// Mitsubishi GX Works2 project: group24_exe2   PLC: FX3G

// global labels: Global1
VAR_GLOBAL
  all_check AT M1 : BOOL;
  switch_check_start AT X007 : BOOL;
  start_day_lamp AT Y007 : BOOL;
  CREAM_CONTAINER AT D2006 : REAL;
  Cream_Transfer_Start AT X011 : BOOL;
  splash_bag AT D2010 : REAL;
  BISCUITS_CONTAINER AT D2012 : REAL;
  Tray AT D2014 : REAL;
  Start_Machine_A AT X010 : BOOL;
  System_On AT M0 : BOOL;
  Close_System AT X005 : BOOL;
  Splashing_System AT Y004 : BOOL;
  Sen1 AT X001 : BOOL;
  Sen4 AT X002 : BOOL;
  Sen30 AT X004 : BOOL;
  Sen15 AT X003 : BOOL;
  Timer_Out_1 AT TS1 : BOOL;
  Sirogin0 AT Y000 : BOOL;
  Sirogin1 AT Y001 : BOOL;
  First_T AT TC1 : BOOL;
  Second_T AT TC2 : BOOL;
  Timer_Out_2 AT TS2 : BOOL;
  Help_Start_1 AT M10 : BOOL;
  Help_Start_2 AT M11 : BOOL;
  Help_Start_3 AT M12 : BOOL;
  Evhov AT M40 : BOOL;
END_VAR
VAR_GLOBAL CONSTANT
  Time_For_Evhov : INT := 40;
END_VAR
VAR_GLOBAL
  start_chocolate AT X006 : BOOL;
END_VAR
VAR_GLOBAL CONSTANT
  input_1 : INT;
  input_5 : INT := 1995;
END_VAR
VAR_GLOBAL
  TC_4 AT TC4 : BOOL;
  Chocolate_Dip_Lamp AT Y003 : BOOL;
  TS_4 AT TS4 : BOOL;
  CRAMBO_PACKAGE_LIGHT AT Y002 : BOOL;
  CC_5 AT CC5 : BOOL;
END_VAR
VAR_GLOBAL CONSTANT
  Count_5 : INT := 5;
END_VAR
VAR_GLOBAL
  CS_5 AT CS5 : BOOL;
  START_PACKAGING AT X000 : BOOL;
  M14_STOP_LAMP AT M14 : BOOL;
END_VAR
VAR_GLOBAL CONSTANT
  Count_6 : INT := 6;
END_VAR
VAR_GLOBAL
  M16_lamp AT M16 : BOOL;
  CS_6 AT CS6 : BOOL;
  CC_6 AT CC6 : BOOL;
END_VAR
VAR_GLOBAL CONSTANT
  input_10 : INT := 4000;
END_VAR
VAR_GLOBAL
  analog_input_10 AT M20 : BOOL;
  analog_input_5 AT M18 : BOOL;
  Check_New_Iteration_Cream AT M24 : BOOL;
  Check_New_Iteration_chocolate AT M26 : BOOL;
  Check_New_Iteration_Biscuits AT M28 : BOOL;
  CHOCOLATE_CONTAINER AT D2022 : REAL;
  CHOCOLATE_DIPPING AT D2020 : REAL;
  TS_30 AT TS30 : BOOL;
  TC_30 AT TC30 : BOOL;
END_VAR
VAR_GLOBAL CONSTANT
  Three_sec : INT := 30;
END_VAR
VAR_GLOBAL
  helperhivhuv AT M9 : BOOL;
  Help_Lamp AT M2 : BOOL;
  analog_input_cream AT D2026 : REAL;
  analog_input_chocolat AT D2028 : REAL;
  analog_input_biscuit AT D2030 : REAL;
  Help_Lamp_On_1 AT M31 : BOOL;
  Help_Lamp_On_2 AT M32 : BOOL;
  Hivhiv_transport AT TC40 : BOOL;
  TS_40 AT TS40 : BOOL;
END_VAR
VAR_GLOBAL CONSTANT
  crembo_mul : REAL := 40;
  const_120 : REAL := 120;
  const_240 : REAL := 240;
  const_300 : REAL := 300;
  const_6 : REAL := 6;
END_VAR
VAR_GLOBAL
  finished_crembos AT D2018 : REAL;
  analogiNPUT AT D8280 : INT;
  save_analogiNPUT AT D2000 : INT;
END_VAR
VAR_GLOBAL CONSTANT
  hivhuv_Seconds : INT := 3;
END_VAR
VAR_GLOBAL
  finished_dipping AT M70 : BOOL;
END_VAR
VAR_GLOBAL CONSTANT
  Timer_For_Chocolate_Dipping : INT := 50;
END_VAR
VAR_GLOBAL
  analog_output AT D8282 : INT;
END_VAR

// task Task_01 (event TRUE, interval 0, priority 31): POU_01

PROGRAM POU_01
(* structured ladder/FBD written out as ST: instructions are called as NAME(EN, inputs, outputs); _pN, _eN, _tN stand for wires *)
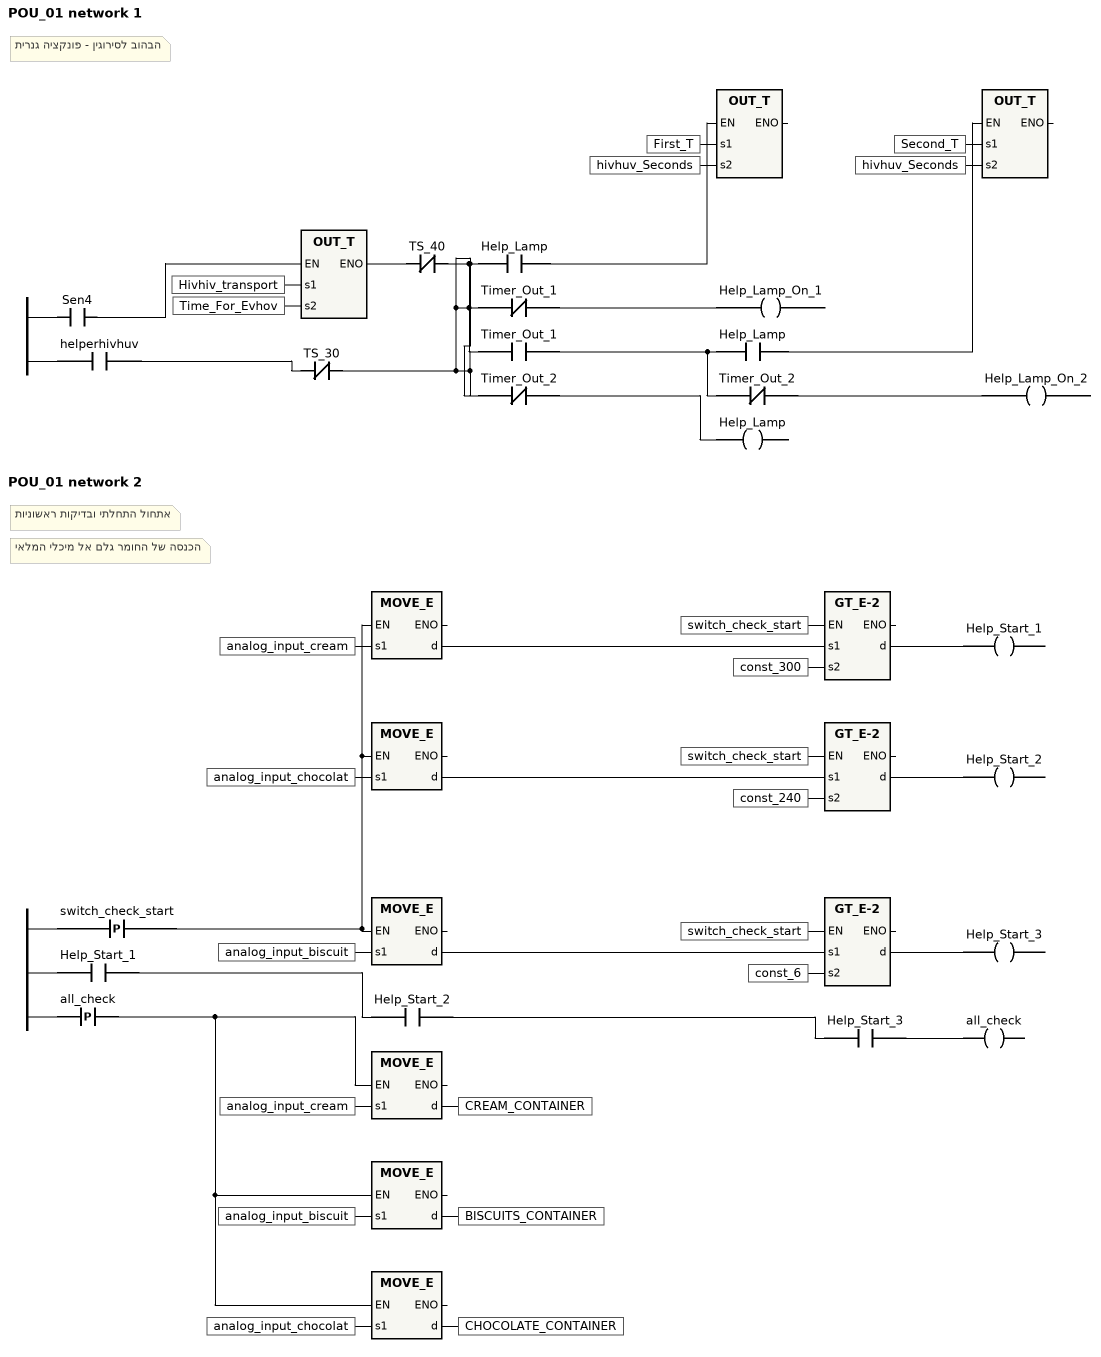
(* network 1 *)
(* הבהוב לסירוגין - פונקציה גנרית *)
_e1 := OUT_T(Sen4, Hivhiv_transport, Time_For_Evhov);
_p2 := (_e1 AND NOT TS_40) OR (helperhivhuv AND NOT TS_30);
OUT_T(_p2 AND Help_Lamp, First_T, hivhuv_Seconds);
Help_Lamp_On_1 := _p2 AND NOT Timer_Out_1;
_p3 := _p2 AND Timer_Out_1;
OUT_T(_p3 AND Help_Lamp, Second_T, hivhuv_Seconds);
Help_Lamp_On_2 := _p3 AND NOT Timer_Out_2;
Help_Lamp := _p2 AND NOT Timer_Out_2;
(* network 2 *)
(* אתחול התחלתי ובדיקות ראשוניות *)
(* הכנסה של החומר גלם אל מיכלי המלאי *)
_p1 := LDP(TRUE, switch_check_start);
MOVE_E(_p1, analog_input_cream, _t2);
GT_E(switch_check_start, _t2, const_300, _t3);
Help_Start_1 := _t3;
MOVE_E(_p1, analog_input_chocolat, _t4);
GT_E(switch_check_start, _t4, const_240, _t5);
Help_Start_2 := _t5;
MOVE_E(_p1, analog_input_biscuit, _t6);
GT_E(switch_check_start, _t6, const_6, _t7);
Help_Start_3 := _t7;
all_check := Help_Start_1 AND Help_Start_2 AND Help_Start_3;
_p8 := LDP(TRUE, all_check);
MOVE_E(_p8, analog_input_cream, CREAM_CONTAINER);
MOVE_E(_p8, analog_input_biscuit, BISCUITS_CONTAINER);
MOVE_E(_p8, analog_input_chocolat, CHOCOLATE_CONTAINER);
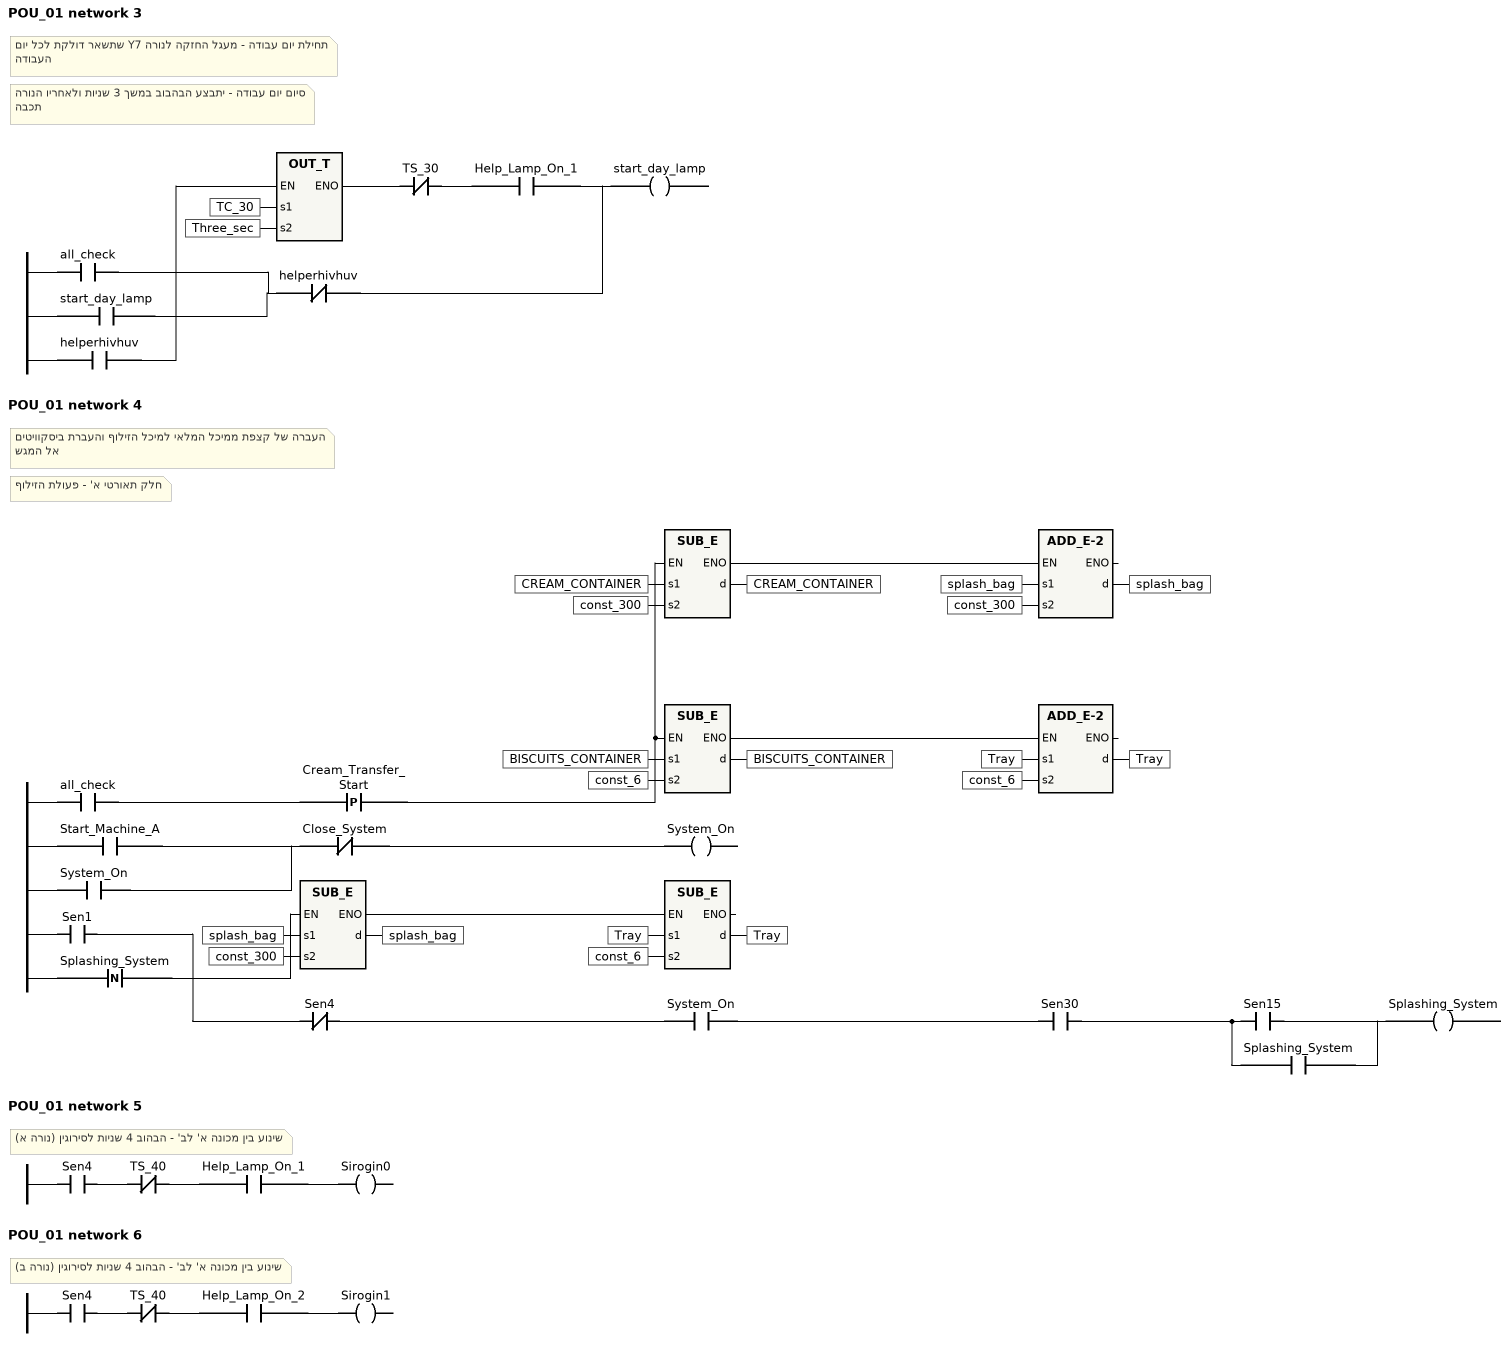
(* network 3 *)
(* תחילת יום עבודה - מעגל החזקה לנורה Y7 שתשאר דולקת לכל יום העבודה *)
(* סיום יום עבודה - יתבצע הבהבוב במשך 3 שניות ולאחריו הנורה תכבה *)
_e1 := OUT_T(helperhivhuv, TC_30, Three_sec);
start_day_lamp := ((all_check OR start_day_lamp) AND NOT helperhivhuv) OR (_e1 AND NOT TS_30 AND Help_Lamp_On_1);
(* network 4 *)
(* העברה של קצפת ממיכל המלאי למיכל הזילוף והעברת ביסקוויטים אל המגש *)
(* חלק תאורטי א' - פעולת הזילוף *)
_p1 := all_check AND LDP(TRUE, Cream_Transfer_Start);
_e2 := SUB_E(_p1, CREAM_CONTAINER, const_300, CREAM_CONTAINER);
ADD_E(_e2, splash_bag, const_300, splash_bag);
_e3 := SUB_E(_p1, BISCUITS_CONTAINER, const_6, BISCUITS_CONTAINER);
ADD_E(_e3, Tray, const_6, Tray);
System_On := (Start_Machine_A OR System_On) AND NOT Close_System;
_p4 := Sen1 AND NOT Sen4 AND System_On AND Sen30;
Splashing_System := (_p4 AND Sen15) OR (_p4 AND Splashing_System);
_e5 := SUB_E(LDF(TRUE, Splashing_System), splash_bag, const_300, splash_bag);
SUB_E(_e5, Tray, const_6, Tray);
(* network 5 *)
(* שינוע בין מכונה א' לב' - הבהוב 4 שניות לסירוגין (נורה א) *)
Sirogin0 := Sen4 AND NOT TS_40 AND Help_Lamp_On_1;
(* network 6 *)
(* שינוע בין מכונה א' לב' - הבהוב 4 שניות לסירוגין (נורה ב) *)
Sirogin1 := Sen4 AND NOT TS_40 AND Help_Lamp_On_2;
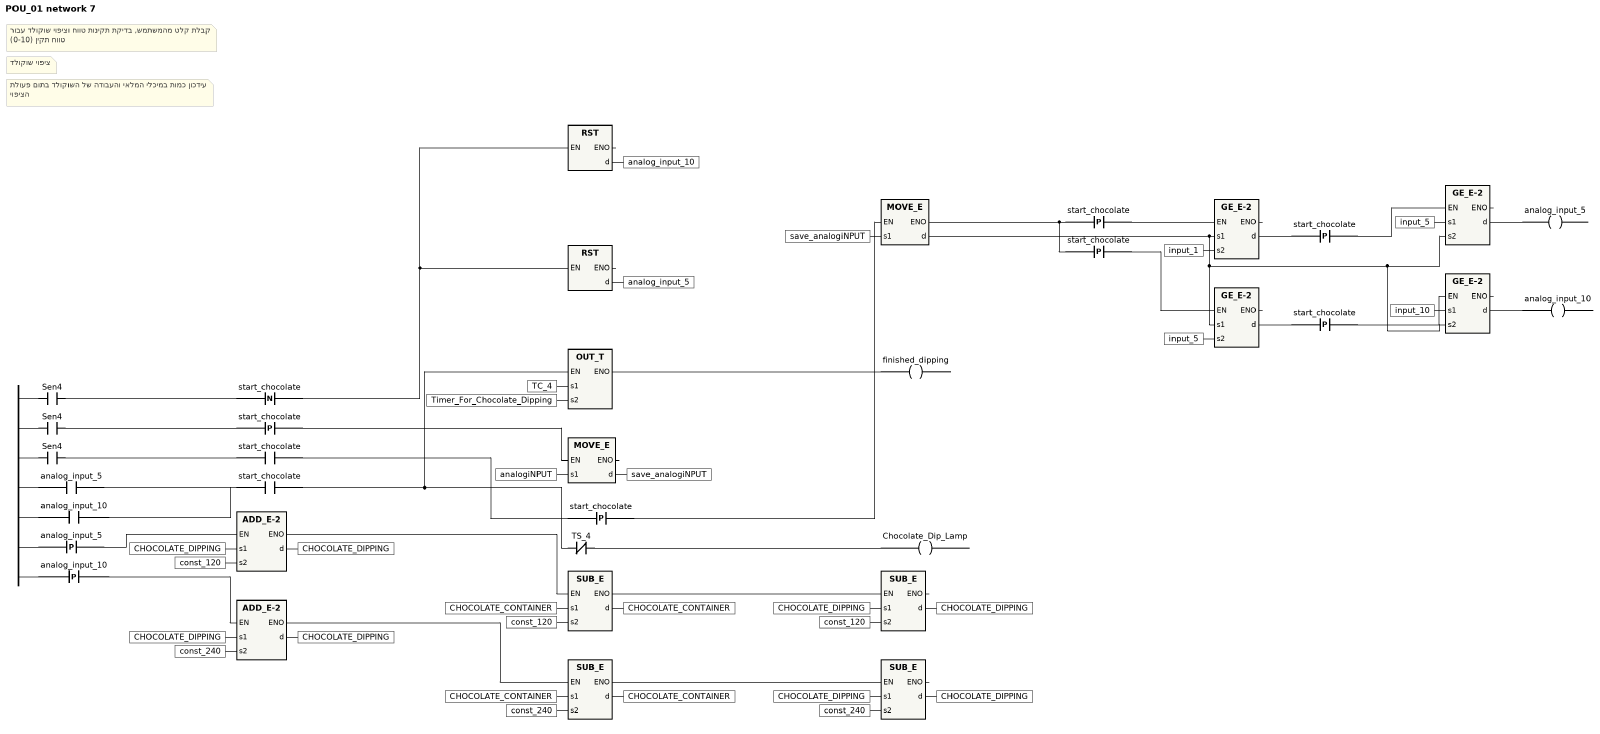
(* network 7 *)
(* קבלת קלט מהמשתמש, בדיקת תקינות טווח וציפוי שוקולד עבור טווח תקין (0-10) *)
(* ציפוי שוקולד *)
(* עידכון כמות במיכלי המלאי והעבודה של השוקולד בתום פעולת הציפוי *)
_p1 := Sen4 AND LDF(TRUE, start_chocolate);
RST(_p1, analog_input_10);
RST(_p1, analog_input_5);
MOVE_E(Sen4 AND LDP(TRUE, start_chocolate), analogiNPUT, save_analogiNPUT);
_e3 := MOVE_E(Sen4 AND start_chocolate AND LDP(TRUE, start_chocolate), save_analogiNPUT, _t2);
GE_E(_e3 AND LDP(TRUE, start_chocolate), _t2, input_1, _t4);
GE_E(_t4 AND LDP(TRUE, start_chocolate), input_5, _t2, _t5);
analog_input_5 := _t5;
GE_E(_e3 AND LDP(TRUE, start_chocolate), _t2, input_5, _t6);
GE_E(_t6 AND LDP(TRUE, start_chocolate), input_10, _t2, _t7);
analog_input_10 := _t7;
_p8 := (analog_input_5 OR analog_input_10) AND start_chocolate;
_e9 := OUT_T(_p8, TC_4, Timer_For_Chocolate_Dipping);
finished_dipping := _e9;
Chocolate_Dip_Lamp := _p8 AND NOT TS_4;
_e10 := ADD_E(LDP(TRUE, analog_input_5), CHOCOLATE_DIPPING, const_120, CHOCOLATE_DIPPING);
_e11 := SUB_E(_e10, CHOCOLATE_CONTAINER, const_120, CHOCOLATE_CONTAINER);
SUB_E(_e11, CHOCOLATE_DIPPING, const_120, CHOCOLATE_DIPPING);
_e12 := ADD_E(LDP(TRUE, analog_input_10), CHOCOLATE_DIPPING, const_240, CHOCOLATE_DIPPING);
_e13 := SUB_E(_e12, CHOCOLATE_CONTAINER, const_240, CHOCOLATE_CONTAINER);
SUB_E(_e13, CHOCOLATE_DIPPING, const_240, CHOCOLATE_DIPPING);
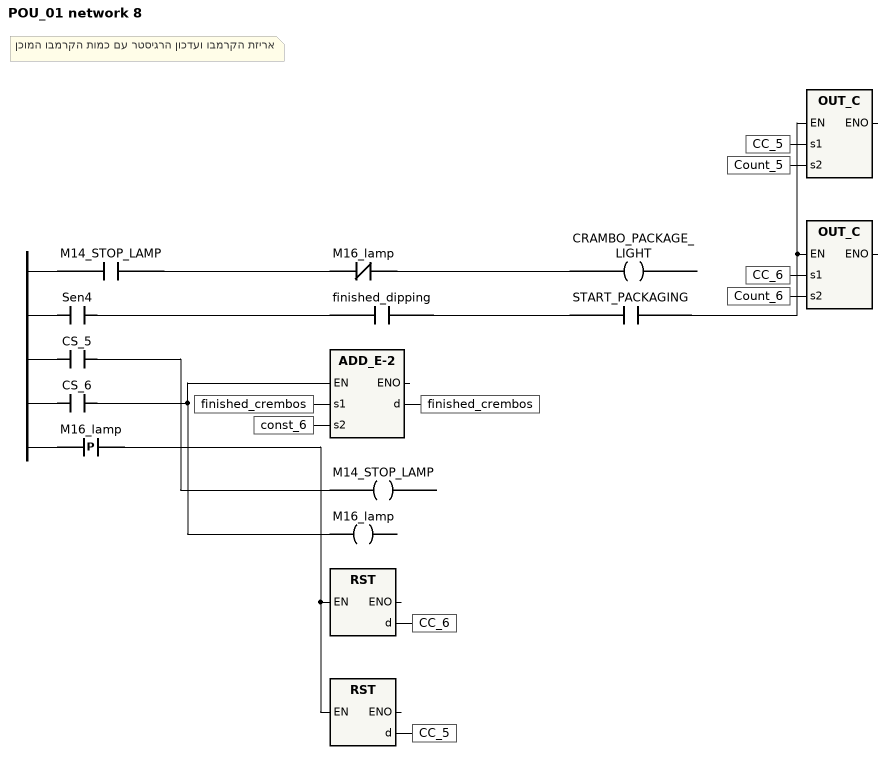
(* network 8 *)
(* אריזת הקרמבו ועדכון הרגיסטר עם כמות הקרמבו המוכן *)
CRAMBO_PACKAGE_LIGHT := M14_STOP_LAMP AND NOT M16_lamp;
_p1 := Sen4 AND finished_dipping AND START_PACKAGING;
OUT_C(_p1, CC_5, Count_5);
OUT_C(_p1, CC_6, Count_6);
M14_STOP_LAMP := CS_5;
M16_lamp := CS_6;
ADD_E(CS_6, finished_crembos, const_6, finished_crembos);
_p2 := LDP(TRUE, M16_lamp);
RST(_p2, CC_6);
RST(_p2, CC_5);
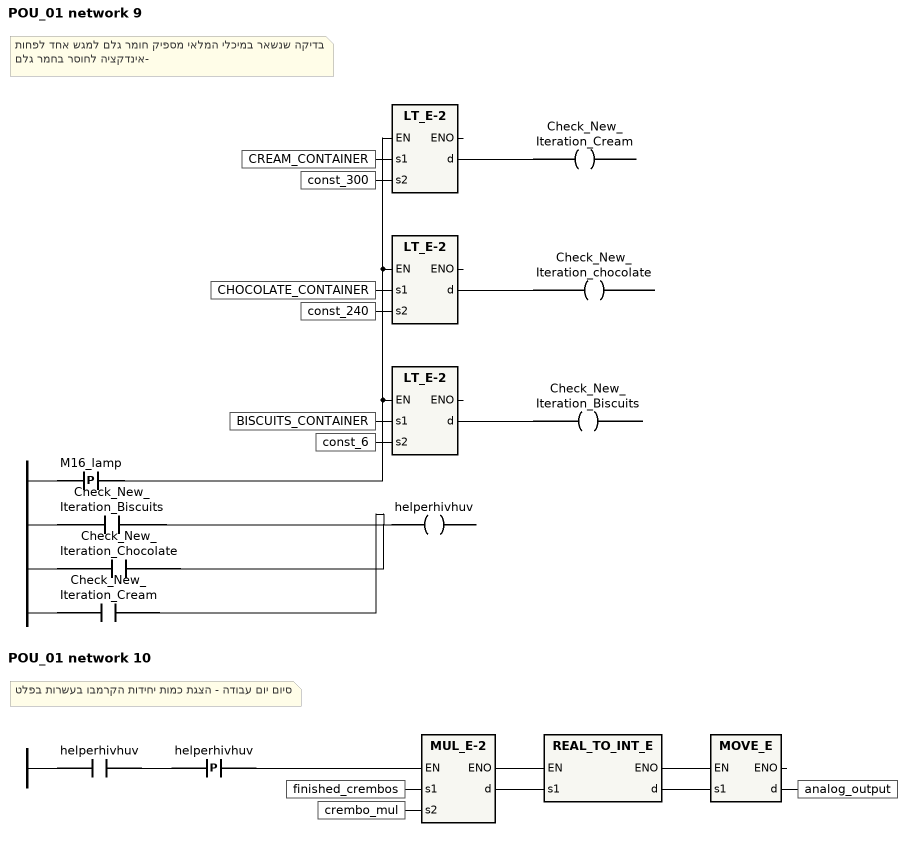
(* network 9 *)
(* בדיקה שנשאר במיכלי המלאי מספיק חומר גלם למגש אחד לפחות -אינדקציה לחוסר בחמר גלם *)
_p1 := LDP(TRUE, M16_lamp);
LT_E(_p1, CREAM_CONTAINER, const_300, _t2);
Check_New_Iteration_Cream := _t2;
LT_E(_p1, CHOCOLATE_CONTAINER, const_240, _t3);
Check_New_Iteration_chocolate := _t3;
LT_E(_p1, BISCUITS_CONTAINER, const_6, _t4);
Check_New_Iteration_Biscuits := _t4;
helperhivhuv := Check_New_Iteration_Biscuits OR Check_New_Iteration_Chocolate OR Check_New_Iteration_Cream;
(* network 10 *)
(* סיום יום עבודה - הצגת כמות יחידות הקרמבו בעשרות בפלט *)
_e2 := MUL_E(helperhivhuv AND LDP(TRUE, helperhivhuv), finished_crembos, crembo_mul, _t1);
_e4 := REAL_TO_INT_E(_e2, _t1, _t3);
MOVE_E(_e4, _t3, analog_output);
END_PROGRAM
